PROGRAM MAIN
VAR
END_VAR

END_PROGRAM

(* stored: Version 1.1.0.1
   POU MAIN: Id {064712f3-f472-4a8d-804d-d85519b6bdbc} *)
